TYPE ST_PositionXY :
STRUCT
	x 		: LREAL;
	Y 		: LREAL;
	valid 	: BOOL;
END_STRUCT
END_TYPE

(* stored: Version 1.1.0.1, ProductVersion 3.1.4024.12
   DUT ST_PositionXY: Id {3382d11b-1e68-4f49-b119-0faea02aae2e} *)
